Staubli VAL3: getYesNo.pgx

public program getYesNo(string& x_sYesNo[])
begin
  x_sYesNo=language:Yes
  x_sYesNo[1]=language:No
end
